CASE fb_state_entry.i16_step OF
	INIT_OBJ:	(* Zylindertyp feststellen *)
		IF st_config.b_config_fertig THEN
			(* Anzahl Spulen *)
			i16_anzahl_spulen := STRING_TO_INT(MID(st_config.str_zylinder_typ, 1, 1));
			(* Anzahl Sensoren *)
			i16_anzahl_sensoren := STRING_TO_INT(MID(st_config.str_zylinder_typ, 1, 3));
			(* Zylinder ist nockengesteuert *)
			IF FIND(st_config.str_zylinder_typ, 'NO') = 0 THEN
				b_nockengesteuert := FALSE;
			ELSE
				b_nockengesteuert := TRUE;
			END_IF
			(* Zylinder ist mit Totzeitkompensation *)
			IF FIND(st_config.str_zylinder_typ, 'TZK') = 0 THEN
				b_mit_tzk := FALSE;
			ELSE
				b_mit_tzk := TRUE;
			END_IF
			(* Vorhandene Sensoren *)
			IF FIND(st_config.str_zylinder_typ, 'AUS') >= 5 THEN
				b_sensor_ausgefahren_vorhanden := TRUE;
			ELSE
				b_sensor_ausgefahren_vorhanden := FALSE;
			END_IF
			IF FIND(st_config.str_zylinder_typ, 'EIN') >= 5 THEN
				b_sensor_eingefahren_vorhanden := TRUE;
			ELSE
				b_sensor_eingefahren_vorhanden := FALSE;
			END_IF
			fb_state_entry.i16_next_step := ZYL_INIT;
		END_IF

(*=======================================================*)
	ZYL_INIT:
		IF fb_state_entry.E THEN
			fb_ton_uz_fahren.IN := FALSE;
			fb_ton_uz_endlage1.IN := FALSE;
			fb_ton_uz_endlage2.IN := FALSE;
			fb_ton_uz_endlage3.IN := FALSE;
			fb_ton_uz_sensor1.IN := FALSE;
			fb_ton_uz_sensor2.IN := FALSE;
			fb_ton_uz_sensor3.IN := FALSE;
			st_tzk.fb_ton_tzk.IN	 := FALSE;
			fb_ton_einausfahren.IN := FALSE;
			fb_ton_quitt.IN := FALSE;
			a_ventil_ausfahren := FALSE;
			a_ventil_einfahren	:= FALSE;
			st_ctrl_out.b_fehler := FALSE;
			st_ctrl_out.b_eingefahren := FALSE;
			st_ctrl_out.b_ausgefahren := FALSE;
			st_ctrl_out.b_gestoppt := FALSE;
			st_ctrl_out.b_ohne_luft := FALSE;
			st_sm.b_zeit_ausfahren1:= FALSE;
			st_sm.b_zeit_einfahren1:= FALSE;
			st_sm.b_endlage1	:= FALSE;
			st_sm.b_sensor1:= FALSE;
			st_sm.b_zeit_ausfahren2 := FALSE;
			st_sm.b_zeit_einfahren2 := FALSE;
			st_sm.b_endlage2	:= FALSE;
			st_sm.b_sensor2 := FALSE;
			st_sm.b_zeit_ausfahren3 := FALSE;
			st_sm.b_zeit_einfahren3 := FALSE;
			st_sm.b_endlage3	:= FALSE;
			st_sm.b_sensor3 := FALSE;
			st_sm.b_winkel_ausfahren1:= FALSE;
			st_sm.b_winkel_einfahren1:= FALSE;
			st_sm.b_winkel_ausfahren2 := FALSE;
			st_sm.b_winkel_einfahren2 := FALSE;
			st_sm.b_winkel_ausfahren3 := FALSE;
			st_sm.b_winkel_einfahren3 := FALSE;
			st_sm.b_zyltyp_nicht_definiert := FALSE;
			st_sm.b_reserve1:= FALSE;
			b_direkttaste_ausfahren := FALSE;
			b_direkttaste_mittefahren := FALSE;
			b_direkttaste_einfahren	 := FALSE;
			b_zustand_uw_nocken_einfahren := FALSE;
			b_zustand_uw_nocken_ausfahren := FALSE;
		END_IF

		(*-----------------------Weiterschaltbedingungen----------------------------*)
		IF e_druckwaechter THEN
			CASE i16_anzahl_sensoren OF
			0:
				fb_state_entry.i16_next_step := GESTOPPT;

			1:
				IF b_nockengesteuert THEN
					IF bw_nocken_zylinder_einfahren THEN
						fb_state_entry.i16_next_step := BEWEGUNG_EINFAHREN;
					ELSIF bw_nocken_zylinder_ausfahren THEN
						fb_state_entry.i16_next_step := BEWEGUNG_AUSFAHREN;
					ELSE
						fb_state_entry.i16_next_step := GESTOPPT;
					END_IF
				ELSE
					IF  b_sensor_ausgefahren_vorhanden THEN
						IF NOT e_sensor1_ausgefahren THEN
							fb_state_entry.i16_next_step := BEWEGUNG_EINFAHREN;
						ELSIF e_sensor1_ausgefahren THEN
							fb_state_entry.i16_next_step := BEWEGUNG_AUSFAHREN;
						ELSE
							fb_state_entry.i16_next_step := GESTOPPT;
						END_IF
					ELSIF  b_sensor_eingefahren_vorhanden THEN
						IF e_sensor1_eingefahren THEN
							fb_state_entry.i16_next_step := BEWEGUNG_EINFAHREN;
						ELSIF NOT e_sensor1_eingefahren THEN
							fb_state_entry.i16_next_step := BEWEGUNG_AUSFAHREN;
						ELSE
							fb_state_entry.i16_next_step := GESTOPPT;
						END_IF
					END_IF
				END_IF

			2:
				IF b_nockengesteuert THEN
					IF bw_nocken_zylinder_einfahren THEN
						fb_state_entry.i16_next_step := BEWEGUNG_EINFAHREN;
					ELSIF bw_nocken_zylinder_ausfahren THEN
						fb_state_entry.i16_next_step := BEWEGUNG_AUSFAHREN;
					ELSE
						fb_state_entry.i16_next_step := GESTOPPT;
					END_IF
				ELSE
					IF b_sensor_eingefahren_vorhanden AND b_sensor_ausgefahren_vorhanden THEN
						IF e_sensor1_eingefahren THEN
							fb_state_entry.i16_next_step := BEWEGUNG_EINFAHREN;
						ELSIF e_sensor1_ausgefahren THEN
							fb_state_entry.i16_next_step := BEWEGUNG_AUSFAHREN;
						ELSE
							fb_state_entry.i16_next_step := GESTOPPT;
						END_IF
					ELSIF b_sensor_ausgefahren_vorhanden THEN
						IF NOT e_sensor1_ausgefahren AND NOT  e_sensor2_ausgefahren THEN
							fb_state_entry.i16_next_step := BEWEGUNG_EINFAHREN;
						ELSIF e_sensor1_ausgefahren OR e_sensor2_ausgefahren THEN
							fb_state_entry.i16_next_step := BEWEGUNG_AUSFAHREN;
						ELSE
							fb_state_entry.i16_next_step := GESTOPPT;
						END_IF
					ELSIF b_sensor_eingefahren_vorhanden THEN
						IF e_sensor1_eingefahren OR  e_sensor2_eingefahren THEN
							fb_state_entry.i16_next_step := BEWEGUNG_EINFAHREN;
						ELSIF NOT e_sensor1_eingefahren AND NOT e_sensor2_eingefahren THEN
							fb_state_entry.i16_next_step := BEWEGUNG_AUSFAHREN;
						ELSE
							fb_state_entry.i16_next_step := GESTOPPT;
						END_IF
					END_IF
				END_IF

			3:
				IF b_nockengesteuert THEN
					IF bw_nocken_zylinder_einfahren THEN
						fb_state_entry.i16_next_step := BEWEGUNG_EINFAHREN;
					ELSIF bw_nocken_zylinder_ausfahren THEN
						fb_state_entry.i16_next_step := BEWEGUNG_AUSFAHREN;
					ELSE
						fb_state_entry.i16_next_step := GESTOPPT;
					END_IF
				ELSE
					IF e_sensor1_eingefahren THEN
						fb_state_entry.i16_next_step := BEWEGUNG_EINFAHREN;
					ELSIF e_sensor1_ausgefahren THEN
						fb_state_entry.i16_next_step := BEWEGUNG_AUSFAHREN;
					ELSE
						fb_state_entry.i16_next_step := GESTOPPT;
					END_IF
				END_IF

			4:
				IF b_nockengesteuert THEN
					IF bw_nocken_zylinder_einfahren THEN
						fb_state_entry.i16_next_step := BEWEGUNG_EINFAHREN;
					ELSIF bw_nocken_zylinder_ausfahren THEN
						fb_state_entry.i16_next_step := BEWEGUNG_AUSFAHREN;
					ELSE
						fb_state_entry.i16_next_step := GESTOPPT;
					END_IF
				ELSE
					IF e_sensor1_eingefahren AND e_sensor2_eingefahren THEN
						fb_state_entry.i16_next_step := BEWEGUNG_EINFAHREN;
					ELSIF e_sensor1_ausgefahren AND e_sensor2_ausgefahren THEN
						fb_state_entry.i16_next_step := BEWEGUNG_AUSFAHREN;
					ELSE
						fb_state_entry.i16_next_step := GESTOPPT;
					END_IF
				END_IF

			6:
				IF b_nockengesteuert THEN
					IF bw_nocken_zylinder_einfahren THEN
						fb_state_entry.i16_next_step := BEWEGUNG_EINFAHREN;
					ELSIF bw_nocken_zylinder_ausfahren THEN
						fb_state_entry.i16_next_step := BEWEGUNG_AUSFAHREN;
					ELSE
						fb_state_entry.i16_next_step := GESTOPPT;
					END_IF
				ELSE
					IF e_sensor1_eingefahren AND e_sensor2_eingefahren AND e_sensor3_eingefahren THEN
						fb_state_entry.i16_next_step := BEWEGUNG_EINFAHREN;
					ELSIF e_sensor1_ausgefahren AND e_sensor2_ausgefahren AND e_sensor3_ausgefahren THEN
						fb_state_entry.i16_next_step := BEWEGUNG_AUSFAHREN;
					ELSE
						fb_state_entry.i16_next_step := GESTOPPT;
					END_IF
				END_IF
			END_CASE
		END_IF

(*=======================================================*)
	GESTOPPT:
		IF fb_state_entry.E THEN
			a_ventil_ausfahren := FALSE;
			a_ventil_einfahren	:= FALSE;
			st_ctrl_out.b_gestoppt := TRUE;
			st_ctrl_out.b_eingefahren := FALSE;
			st_ctrl_out.b_ausgefahren := FALSE;
			st_ctrl_out.b_ohne_luft := FALSE;
			st_ctrl_out.b_fehler := FALSE;
			b_zustand_uw_nocken_einfahren := FALSE;
			b_zustand_uw_nocken_ausfahren := FALSE;
		END_IF

		(*-----------------------Weiterschaltbedingungen----------------------------*)
		CASE i16_betriebsart OF
		KEINE:
			;
		AUTO, TIPPEN, DUMMY, PSEUDO:
			IF 	(st_ctrl_in.b_ausfahren AND
				NOT bw_nocken_zylinder_ausfahren AND
				NOT b_ibn_zylinder_ausfahren AND
				NOT b_direkttaste_ausfahren AND
				NOT e_taste_ausfahren) OR
				(NOT st_ctrl_in.b_ausfahren AND
				bw_nocken_zylinder_ausfahren AND
				NOT b_ibn_zylinder_ausfahren AND
				NOT b_direkttaste_ausfahren AND
				NOT e_taste_ausfahren) OR
				(NOT st_ctrl_in.b_ausfahren AND
				NOT bw_nocken_zylinder_ausfahren AND
				b_ibn_zylinder_ausfahren AND
				NOT b_direkttaste_ausfahren AND
				NOT e_taste_ausfahren)
				THEN
					fb_state_entry.i16_next_step := BEWEGUNG_AUSFAHREN;

			ELSIF	(st_ctrl_in.b_einfahren AND
					NOT bw_nocken_zylinder_einfahren AND
					NOT b_ibn_zylinder_einfahren AND
					NOT b_direkttaste_einfahren AND
					NOT e_taste_einfahren) OR
					(NOT st_ctrl_in.b_einfahren AND
					bw_nocken_zylinder_einfahren AND
					NOT b_ibn_zylinder_einfahren AND
					NOT b_direkttaste_einfahren AND
					NOT e_taste_einfahren) OR
					(NOT st_ctrl_in.b_einfahren AND
					NOT bw_nocken_zylinder_einfahren AND
					b_ibn_zylinder_einfahren AND
					NOT b_direkttaste_einfahren AND
					NOT e_taste_einfahren)
					THEN
						fb_state_entry.i16_next_step := BEWEGUNG_EINFAHREN;

			ELSIF	st_ctrl_in.b_luftlos AND
					NOT bw_nocken_zylinder_einfahren AND
					NOT b_ibn_zylinder_einfahren AND
					NOT b_direkttaste_einfahren AND
					NOT e_taste_einfahren AND
					NOT bw_nocken_zylinder_ausfahren AND
					NOT b_ibn_zylinder_ausfahren AND
					NOT b_direkttaste_ausfahren AND
					NOT e_taste_ausfahren
					THEN
						fb_state_entry.i16_next_step := LUFTLOS;
			END_IF
		HAND:
			IF	(st_visu.i16_nr_zyl_im_handbetrieb = st_config.i16_identnummer AND (st_visu.b_taste_ausfahren OR e_taste_ausfahren)) OR
				(bw_nocken_zylinder_ausfahren AND b_nockengesteuert AND b_masterachse_hand_dialog_aktiv)
				THEN
					fb_state_entry.i16_next_step := BEWEGUNG_AUSFAHREN;

			ELSIF	(st_visu.i16_nr_zyl_im_handbetrieb = st_config.i16_identnummer AND (st_visu.b_taste_einfahren OR e_taste_einfahren)) OR
					(bw_nocken_zylinder_einfahren AND b_nockengesteuert AND b_masterachse_hand_dialog_aktiv)
					THEN
						fb_state_entry.i16_next_step := BEWEGUNG_EINFAHREN;
			END_IF
		END_CASE

(*=======================================================*)
	EINGEFAHREN:
		IF fb_state_entry.E THEN
			st_ctrl_out.b_gestoppt := FALSE;
			st_ctrl_out.b_ausgefahren := FALSE;
			st_ctrl_out.b_ohne_luft := FALSE;
			fb_ton_einausfahren.IN := FALSE;
			fb_ton_uz_fahren.IN := FALSE;
			fb_ton_uz_sensor1.IN := FALSE;
			fb_ton_uz_sensor2.IN := FALSE;
			fb_ton_uz_sensor3.IN := FALSE;
			st_tzk.fb_ton_tzk.IN := FALSE;
			a_ventil_einfahren := TRUE;
			b_zustand_uw_nocken_einfahren := FALSE;
			IF NOT b_mit_tzk THEN
				st_ctrl_out.b_eingefahren := TRUE;
			END_IF
		END_IF

		IF st_ctrl_in.b_einfahren THEN	(* Messagewiederholung wenn der Zylinder sich schon im gewünschten Zustand befindet*)
			st_ctrl_out.b_eingefahren := TRUE;
		END_IF
	
		(*-----------------------Weiterschaltbedingungen----------------------------*)
		CASE i16_betriebsart OF
		KEINE:
			;
		AUTO, TIPPEN, DUMMY, PSEUDO:
			IF 	(st_ctrl_in.b_ausfahren AND
				NOT bw_nocken_zylinder_ausfahren AND
				NOT b_ibn_zylinder_ausfahren AND
				NOT b_direkttaste_ausfahren AND
				NOT e_taste_ausfahren) OR
				(NOT st_ctrl_in.b_ausfahren AND
				bw_nocken_zylinder_ausfahren  AND
				NOT b_ibn_zylinder_ausfahren AND
				NOT b_direkttaste_ausfahren AND
				NOT e_taste_ausfahren) OR
				(NOT st_ctrl_in.b_ausfahren AND
				NOT bw_nocken_zylinder_ausfahren AND
				b_ibn_zylinder_ausfahren AND
				NOT b_direkttaste_ausfahren AND
				NOT e_taste_ausfahren)
				THEN
					IF i16_anzahl_sensoren >= 1AND b_sensor_ausgefahren_vorhanden AND b_mit_tzk THEN
						st_tzk.t_ausfahrzeit_kompensiert := (st_tzk.t_ausfahrzeit * st_config.i16_tzk_faktor_ausfahren) / 100;
					END_IF
					fb_state_entry.i16_next_step := BEWEGUNG_AUSFAHREN;

			ELSIF	st_ctrl_in.b_luftlos AND
					NOT bw_nocken_zylinder_einfahren AND
					NOT b_ibn_zylinder_einfahren AND
					NOT b_direkttaste_einfahren AND
					NOT e_taste_einfahren AND
					NOT bw_nocken_zylinder_ausfahren AND
					NOT b_ibn_zylinder_ausfahren AND
					NOT b_direkttaste_ausfahren AND
					NOT e_taste_ausfahren
					THEN
						fb_state_entry.i16_next_step := LUFTLOS;
			END_IF
		HAND:
			IF	(st_visu.i16_nr_zyl_im_handbetrieb = st_config.i16_identnummer AND (st_visu.b_taste_ausfahren OR e_taste_ausfahren)) OR
				(bw_nocken_zylinder_ausfahren AND b_nockengesteuert AND b_masterachse_hand_dialog_aktiv)
				THEN
					IF i16_anzahl_sensoren >= 1AND b_sensor_ausgefahren_vorhanden AND b_mit_tzk THEN
						st_tzk.t_ausfahrzeit_kompensiert := (st_tzk.t_ausfahrzeit * st_config.i16_tzk_faktor_ausfahren) / 100;
					END_IF
					fb_state_entry.i16_next_step := BEWEGUNG_AUSFAHREN;
			END_IF
		END_CASE

		(* Überwachung auf Endlagenfehler *)
		IF i16_betriebsart <> HAND AND st_config.b_aktiv THEN
			CASE i16_anzahl_sensoren OF
				1,2,3:	(* Alle Zylinder mit mindestens einem Sensor für EINGEFAHREN *)
					IF b_sensor_eingefahren_vorhanden AND	st_config.b_endlage1_aktiv AND NOT e_sensor1_eingefahren THEN
						fb_ton_uz_endlage1.IN := TRUE;
						IF fb_ton_uz_endlage1.Q THEN
							st_sm.b_endlage1 := TRUE;
							fb_state_entry.i16_next_step := ZYL_FEHLER;
						END_IF
					ELSE
						fb_ton_uz_endlage1.IN := FALSE;
					END_IF
	
				4:	(* Alle Zylinder mit 2 Sensoren für EINGEFAHREN *)
					IF b_sensor_eingefahren_vorhanden AND st_config.b_endlage1_aktiv AND NOT e_sensor1_eingefahren THEN
						fb_ton_uz_endlage1.IN := TRUE;
						IF fb_ton_uz_endlage1.Q THEN
							st_sm.b_endlage1 := TRUE;
							fb_state_entry.i16_next_step := ZYL_FEHLER;
						END_IF
					ELSE
						fb_ton_uz_endlage1.IN := FALSE;
					END_IF
					IF b_sensor_eingefahren_vorhanden AND st_config.b_endlage2_aktiv AND NOT e_sensor2_eingefahren THEN
						fb_ton_uz_endlage2.IN := TRUE;
						IF fb_ton_uz_endlage2.Q THEN
							st_sm.b_endlage2 := TRUE;
							fb_state_entry.i16_next_step := ZYL_FEHLER;
						END_IF
					ELSE
						fb_ton_uz_endlage2.IN := FALSE;
					END_IF
	
				6:	(* Alle Zylinder mit 3 Sensoren für EINGEFAHREN *)
					IF b_sensor_eingefahren_vorhanden AND st_config.b_endlage1_aktiv AND NOT e_sensor1_eingefahren THEN
						fb_ton_uz_endlage1.IN := TRUE;
						IF fb_ton_uz_endlage1.Q THEN
							st_sm.b_endlage1 := TRUE;
							fb_state_entry.i16_next_step := ZYL_FEHLER;
						END_IF
					ELSE
						fb_ton_uz_endlage1.IN := FALSE;
					END_IF
					IF b_sensor_eingefahren_vorhanden AND st_config.b_endlage2_aktiv AND NOT e_sensor2_eingefahren THEN
						fb_ton_uz_endlage2.IN := TRUE;
						IF fb_ton_uz_endlage2.Q THEN
							st_sm.b_endlage2 := TRUE;
							fb_state_entry.i16_next_step := ZYL_FEHLER;
						END_IF
					ELSE
						fb_ton_uz_endlage2.IN := FALSE;
					END_IF
					IF b_sensor_eingefahren_vorhanden AND st_config.b_endlage3_aktiv AND NOT e_sensor3_eingefahren THEN
						fb_ton_uz_endlage3.IN := TRUE;
						IF fb_ton_uz_endlage3.Q THEN
							st_sm.b_endlage3 := TRUE;
							fb_state_entry.i16_next_step := ZYL_FEHLER;
						END_IF
					ELSE
						fb_ton_uz_endlage3.IN := FALSE;
					END_IF
			END_CASE
		END_IF

(*=======================================================*)
	BEWEGUNG_AUSFAHREN:
		IF fb_state_entry.E THEN
			st_ctrl_out.b_gestoppt := FALSE;
			st_ctrl_out.b_eingefahren := FALSE;
			st_ctrl_out.b_ausgefahren := FALSE;
			st_ctrl_out.b_ohne_luft := FALSE;
			st_ctrl_out.b_fehler := FALSE;
			a_ventil_einfahren := FALSE;
			a_ventil_ausfahren := TRUE;
			fb_ton_uz_fahren.IN := TRUE;
			fb_ton_einausfahren.IN := TRUE;
			fb_ton_uz_endlage1.IN := FALSE;
			fb_ton_uz_endlage2.IN := FALSE;
			fb_ton_uz_endlage3.IN := FALSE;
			st_sm.b_zeit_ausfahren1:= FALSE;
			st_sm.b_zeit_einfahren1:= FALSE;
			st_sm.b_endlage1	:= FALSE;
			st_sm.b_sensor1:= FALSE;
			st_sm.b_zeit_ausfahren2 := FALSE;
			st_sm.b_zeit_einfahren2 := FALSE;
			st_sm.b_endlage2	:= FALSE;
			st_sm.b_sensor2 := FALSE;
			st_sm.b_zeit_ausfahren3 := FALSE;
			st_sm.b_zeit_einfahren3 := FALSE;
			st_sm.b_endlage3	:= FALSE;
			st_sm.b_sensor3 := FALSE;
			st_sm.b_winkel_ausfahren1:= FALSE;
			st_sm.b_winkel_einfahren1:= FALSE;
			st_sm.b_winkel_ausfahren2 := FALSE;
			st_sm.b_winkel_einfahren2 := FALSE;
			st_sm.b_winkel_ausfahren3 := FALSE;
			st_sm.b_winkel_einfahren3 := FALSE;
			st_sm.b_zyltyp_nicht_definiert := FALSE;
			st_sm.b_reserve1:= FALSE;
			(* Verhindere die sofortige Fehlerauslösung, wenn Überwachungsnocken bei Stateentry schon vorhanden ist *)
			IF uw_nocken_zylinder_ausfahren THEN
				b_zustand_uw_nocken_ausfahren := TRUE;
			END_IF
		END_IF

		(* Fehlermeldung für nockengesteuerte Zylinder wieder freischalten *)
		IF fb_ton_uz_fahren.Q THEN
			b_zustand_uw_nocken_ausfahren := FALSE;
		END_IF

		CASE i16_betriebsart OF
		KEINE:
			;
		AUTO, TIPPEN, DUMMY, PSEUDO:
			IF	(st_ctrl_in.b_einfahren AND
				NOT bw_nocken_zylinder_einfahren AND
				NOT b_ibn_zylinder_einfahren AND
				NOT b_direkttaste_einfahren AND
				NOT e_taste_einfahren) OR
				(NOT st_ctrl_in.b_einfahren AND
				bw_nocken_zylinder_einfahren AND
				NOT b_ibn_zylinder_einfahren AND
				NOT b_direkttaste_einfahren AND
				NOT e_taste_einfahren) OR
				(NOT st_ctrl_in.b_einfahren AND
				NOT bw_nocken_zylinder_einfahren AND
				b_ibn_zylinder_einfahren AND
				NOT b_direkttaste_einfahren AND
				NOT e_taste_einfahren)
				THEN
					IF i16_anzahl_sensoren >= 1AND b_sensor_eingefahren_vorhanden AND b_mit_tzk THEN
						st_tzk.t_einfahrzeit_kompensiert := (st_tzk.t_einfahrzeit * st_config.i16_tzk_faktor_einfahren) / 100;
					END_IF
					fb_state_entry.i16_next_step := BEWEGUNG_EINFAHREN;
			END_IF
		HAND:
			IF	(st_visu.i16_nr_zyl_im_handbetrieb = st_config.i16_identnummer AND (st_visu.b_taste_einfahren OR e_taste_einfahren)) OR
				(bw_nocken_zylinder_einfahren AND b_nockengesteuert AND b_masterachse_hand_dialog_aktiv)
				THEN
					IF i16_anzahl_sensoren >= 1AND b_sensor_eingefahren_vorhanden AND b_mit_tzk THEN
						st_tzk.t_einfahrzeit_kompensiert := (st_tzk.t_einfahrzeit * st_config.i16_tzk_faktor_einfahren) / 100;
					END_IF
					fb_state_entry.i16_next_step := BEWEGUNG_EINFAHREN;
			END_IF
		END_CASE

		(* Totzeitkompensation mit Plausibilitätscheck der ermittelten Kompensationszeit *)
		IF	i16_anzahl_sensoren >= 1AND
			b_mit_tzk AND
			b_sensor_ausgefahren_vorhanden AND
			st_tzk.t_ausfahrzeit_kompensiert < st_tzk.t_ausfahrzeit
			THEN
				st_tzk.fb_ton_tzk.PT := st_tzk.t_ausfahrzeit_kompensiert ;
				st_tzk.fb_ton_tzk.IN := TRUE;
				(* Totzeit ist abgelaufen -> vorzeitig "ausgefahren" melden*)
				IF st_tzk.fb_ton_tzk.Q THEN
					st_ctrl_out.b_ausgefahren := TRUE;
				END_IF
		END_IF

		(*-----------------------Weiterschaltbedingungen----------------------------*)
		(* Bedingungen für Zylinder ist ausgefahren und Fehlervorkommen*)
		(* Die Sensorkonfiguration "vorhanden" ist nur für die Fälle 1, 2 von Bedeutung wegen Sonderzylinder *)
		CASE i16_anzahl_sensoren OF
			0:
				IF fb_ton_einausfahren.Q THEN
					fb_state_entry.i16_next_step := AUSGEFAHREN;
				END_IF

			1:
				IF b_sensor_ausgefahren_vorhanden THEN
					IF e_sensor1_ausgefahren THEN
						fb_state_entry.i16_next_step := AUSGEFAHREN;
					ELSE
						IF i16_betriebsart <> HAND AND st_config.b_aktiv THEN
							(* Zeitüberwachung *)
							IF fb_ton_uz_fahren.Q AND (NOT b_nockengesteuert OR b_no_gesteuert_im_norm_betrieb) THEN
								st_sm.b_zeit_ausfahren1 := TRUE;
								fb_state_entry.i16_next_step := ZYL_FEHLER;
							(* Winkelüberwachung *)
							ELSIF uw_nocken_zylinder_ausfahren AND b_nockengesteuert AND NOT b_no_gesteuert_im_norm_betrieb AND NOT b_zustand_uw_nocken_ausfahren THEN
								st_sm.b_winkel_ausfahren1 := TRUE;
								fb_state_entry.i16_next_step := ZYL_FEHLER;
							END_IF
						END_IF
					END_IF
				ELSIF b_sensor_eingefahren_vorhanden THEN
					IF  NOT e_sensor1_eingefahren THEN
						fb_state_entry.i16_next_step := AUSGEFAHREN;
					ELSE
						IF i16_betriebsart <> HAND AND st_config.b_aktiv THEN
							(* Zeitüberwachung *)
							IF fb_ton_uz_fahren.Q AND (NOT b_nockengesteuert OR b_no_gesteuert_im_norm_betrieb) THEN
								st_sm.b_zeit_ausfahren1 := TRUE;
								fb_state_entry.i16_next_step := ZYL_FEHLER;
							(* Winkelüberwachung *)
							ELSIF uw_nocken_zylinder_ausfahren AND b_nockengesteuert AND NOT b_no_gesteuert_im_norm_betrieb AND NOT b_zustand_uw_nocken_ausfahren THEN
								st_sm.b_winkel_ausfahren1 := TRUE;
								fb_state_entry.i16_next_step := ZYL_FEHLER;
							END_IF
						END_IF
					END_IF
				END_IF

			2:
				IF b_sensor_eingefahren_vorhanden AND b_sensor_ausgefahren_vorhanden THEN
					IF e_sensor1_ausgefahren AND NOT e_sensor1_eingefahren THEN
						fb_state_entry.i16_next_step := AUSGEFAHREN;
					ELSE
						IF i16_betriebsart <> HAND AND st_config.b_aktiv THEN
							(* Zeitüberwachung *)
							IF fb_ton_uz_fahren.Q AND (NOT b_nockengesteuert OR b_no_gesteuert_im_norm_betrieb) THEN
								st_sm.b_zeit_ausfahren1 := TRUE;
								fb_state_entry.i16_next_step := ZYL_FEHLER;
							(* Winkelüberwachung *)
							ELSIF uw_nocken_zylinder_ausfahren AND b_nockengesteuert AND NOT b_no_gesteuert_im_norm_betrieb AND NOT b_zustand_uw_nocken_ausfahren THEN
								st_sm.b_winkel_ausfahren1 := TRUE;
								fb_state_entry.i16_next_step := ZYL_FEHLER;
							END_IF
						END_IF
					END_IF
				ELSIF b_sensor_eingefahren_vorhanden THEN
					IF NOT e_sensor1_eingefahren AND NOT e_sensor2_eingefahren THEN
						fb_state_entry.i16_next_step := AUSGEFAHREN;
					ELSE
						IF i16_betriebsart <> HAND AND st_config.b_aktiv THEN
							(* Zeitüberwachung *)
							IF fb_ton_uz_fahren.Q AND (NOT b_nockengesteuert OR b_no_gesteuert_im_norm_betrieb) THEN
								IF e_sensor1_eingefahren THEN
									st_sm.b_zeit_ausfahren1 := TRUE;
								END_IF
								IF e_sensor2_eingefahren THEN
									st_sm.b_zeit_ausfahren2 := TRUE;
								END_IF
								fb_state_entry.i16_next_step := ZYL_FEHLER;
							(* Winkelüberwachung *)
							ELSIF uw_nocken_zylinder_ausfahren AND b_nockengesteuert AND NOT b_no_gesteuert_im_norm_betrieb AND NOT b_zustand_uw_nocken_ausfahren THEN
								IF e_sensor1_eingefahren THEN
									st_sm.b_winkel_ausfahren1 := TRUE;
								END_IF
								IF e_sensor2_eingefahren THEN
									st_sm.b_winkel_ausfahren2 := TRUE;
								END_IF
								fb_state_entry.i16_next_step := ZYL_FEHLER;
							END_IF
						END_IF
					END_IF
				ELSIF  b_sensor_ausgefahren_vorhanden THEN
					IF e_sensor1_ausgefahren AND e_sensor2_ausgefahren THEN
						fb_state_entry.i16_next_step := AUSGEFAHREN;
					ELSE
						IF i16_betriebsart <> HAND AND st_config.b_aktiv THEN
							(* Zeitüberwachung *)
							IF fb_ton_uz_fahren.Q AND (NOT b_nockengesteuert OR b_no_gesteuert_im_norm_betrieb) THEN
								IF NOT e_sensor1_ausgefahren THEN
									st_sm.b_zeit_ausfahren1 := TRUE;
								END_IF
								IF NOT e_sensor2_ausgefahren THEN
									st_sm.b_zeit_ausfahren2 := TRUE;
								END_IF
								fb_state_entry.i16_next_step := ZYL_FEHLER;
							(* Winkelüberwachung *)
							ELSIF uw_nocken_zylinder_ausfahren AND b_nockengesteuert AND NOT b_no_gesteuert_im_norm_betrieb AND NOT b_zustand_uw_nocken_ausfahren THEN
								IF NOT e_sensor1_ausgefahren THEN
									st_sm.b_winkel_ausfahren1 := TRUE;
								END_IF
								IF NOT e_sensor2_ausgefahren THEN
									st_sm.b_winkel_ausfahren2 := TRUE;
								END_IF
								fb_state_entry.i16_next_step := ZYL_FEHLER;
							END_IF
						END_IF
					END_IF
				END_IF
				IF i16_betriebsart <> HAND AND st_config.b_aktiv THEN
					(* Überwachung auf Sensorfehler *)
					IF e_sensor1_ausgefahren  AND e_sensor1_eingefahren  AND st_config.b_sensor1_aktiv THEN
						fb_ton_uz_sensor1.IN := TRUE;
						IF fb_ton_uz_sensor1.Q THEN
							st_sm.b_sensor1 := TRUE;
							fb_state_entry.i16_next_step := ZYL_FEHLER;
						END_IF
					ELSE
						fb_ton_uz_sensor1.IN := FALSE;
					END_IF
				END_IF

			3:
				IF	(* Zylinder ist ausgefahren *)
					(e_sensor1_ausgefahren AND NOT e_sensor1_eingefahren AND NOT e_sensor_mittegefahren) OR
					(* Zylinder steht in Mittelstellung *)
					(e_sensor_mittegefahren AND NOT e_sensor1_eingefahren AND NOT e_sensor1_ausgefahren)
					THEN
						fb_state_entry.i16_next_step := AUSGEFAHREN;
				ELSE
					IF i16_betriebsart <> HAND AND st_config.b_aktiv THEN
						(* Zeitüberwachung *)
						IF fb_ton_uz_fahren.Q AND (NOT b_nockengesteuert OR b_no_gesteuert_im_norm_betrieb) THEN
							st_sm.b_zeit_ausfahren1 := TRUE;
							fb_state_entry.i16_next_step := ZYL_FEHLER;
						(* Winkelüberwachung *)
						ELSIF uw_nocken_zylinder_ausfahren AND b_nockengesteuert AND NOT b_no_gesteuert_im_norm_betrieb AND NOT b_zustand_uw_nocken_ausfahren THEN
							st_sm.b_winkel_ausfahren1 := TRUE;
							fb_state_entry.i16_next_step := ZYL_FEHLER;
						END_IF
					END_IF
				END_IF
				IF i16_betriebsart <> HAND AND st_config.b_aktiv THEN
					(* Überwachung auf Sensorfehler *)
					IF e_sensor1_ausgefahren  AND e_sensor1_eingefahren  AND st_config.b_sensor1_aktiv THEN
						fb_ton_uz_sensor1.IN := TRUE;
						IF fb_ton_uz_sensor1.Q THEN
							st_sm.b_sensor1 := TRUE;
							fb_state_entry.i16_next_step := ZYL_FEHLER;
						END_IF
					ELSE
						fb_ton_uz_sensor1.IN := FALSE;
					END_IF
				END_IF

			4:
				IF e_sensor1_ausgefahren AND e_sensor2_ausgefahren AND NOT e_sensor1_eingefahren AND NOT e_sensor2_eingefahren	THEN
					fb_state_entry.i16_next_step := AUSGEFAHREN;
				ELSE
					IF i16_betriebsart <> HAND AND st_config.b_aktiv THEN
						IF NOT e_sensor1_ausgefahren OR NOT e_sensor2_ausgefahren THEN
							(* Zeitüberwachung *)
							IF fb_ton_uz_fahren.Q AND (NOT b_nockengesteuert OR b_no_gesteuert_im_norm_betrieb) THEN
								IF NOT e_sensor1_ausgefahren THEN
									st_sm.b_zeit_ausfahren1 := TRUE;
								END_IF
								IF NOT e_sensor2_ausgefahren THEN
									st_sm.b_zeit_ausfahren2 := TRUE;
								END_IF
								fb_state_entry.i16_next_step := ZYL_FEHLER;
							(* Winkelüberwachung *)
							ELSIF uw_nocken_zylinder_ausfahren AND b_nockengesteuert AND NOT b_no_gesteuert_im_norm_betrieb AND NOT b_zustand_uw_nocken_ausfahren THEN
								IF NOT e_sensor1_ausgefahren THEN
									st_sm.b_winkel_ausfahren1 := TRUE;
								END_IF
								IF NOT e_sensor2_ausgefahren THEN
									st_sm.b_winkel_ausfahren2 := TRUE;
								END_IF
								fb_state_entry.i16_next_step := ZYL_FEHLER;
							END_IF
						END_IF
					END_IF
				END_IF

				IF i16_betriebsart <> HAND AND st_config.b_aktiv THEN
					(* Überwachung auf Sensorfehler *)
					IF e_sensor1_ausgefahren  AND e_sensor1_eingefahren  AND st_config.b_sensor1_aktiv THEN
						fb_ton_uz_sensor1.IN := TRUE;
						IF fb_ton_uz_sensor1.Q THEN
							st_sm.b_sensor1 := TRUE;
							fb_state_entry.i16_next_step := ZYL_FEHLER;
						END_IF
					ELSE
						fb_ton_uz_sensor1.IN := FALSE;
					END_IF
					IF e_sensor2_ausgefahren  AND e_sensor2_eingefahren  AND st_config.b_sensor2_aktiv THEN
						fb_ton_uz_sensor2.IN := TRUE;
						IF fb_ton_uz_sensor2.Q THEN
							st_sm.b_sensor2 := TRUE;
							fb_state_entry.i16_next_step := ZYL_FEHLER;
						END_IF
					ELSE
						fb_ton_uz_sensor2.IN := FALSE;
					END_IF
				END_IF

			6:
				IF 	e_sensor1_ausgefahren AND
					e_sensor2_ausgefahren AND
					e_sensor3_ausgefahren AND
					NOT e_sensor1_eingefahren AND
					NOT e_sensor2_eingefahren AND
					NOT e_sensor3_eingefahren
					THEN
						fb_state_entry.i16_next_step := AUSGEFAHREN;
				ELSE
					IF i16_betriebsart <> HAND AND st_config.b_aktiv THEN
						IF NOT e_sensor1_ausgefahren OR NOT e_sensor2_ausgefahren OR NOT e_sensor3_ausgefahren THEN
							(* Zeitüberwachung *)
							IF fb_ton_uz_fahren.Q AND (NOT b_nockengesteuert OR b_no_gesteuert_im_norm_betrieb) THEN
								IF NOT e_sensor1_ausgefahren THEN
									st_sm.b_zeit_ausfahren1 := TRUE;
								END_IF
								IF NOT e_sensor2_ausgefahren THEN
									st_sm.b_zeit_ausfahren2 := TRUE;
								END_IF
								IF NOT e_sensor3_ausgefahren THEN
									st_sm.b_zeit_ausfahren3 := TRUE;
								END_IF
								fb_state_entry.i16_next_step := ZYL_FEHLER;
							(* Winkelüberwachung *)
							ELSIF uw_nocken_zylinder_ausfahren AND b_nockengesteuert AND NOT b_no_gesteuert_im_norm_betrieb AND NOT b_zustand_uw_nocken_ausfahren THEN
								IF NOT e_sensor1_ausgefahren THEN
									st_sm.b_winkel_ausfahren1 := TRUE;
								END_IF
								IF NOT e_sensor2_ausgefahren THEN
									st_sm.b_winkel_ausfahren2 := TRUE;
								END_IF
								IF NOT e_sensor3_ausgefahren THEN
									st_sm.b_winkel_ausfahren3 := TRUE;
								END_IF
								fb_state_entry.i16_next_step := ZYL_FEHLER;
							END_IF
						END_IF
					END_IF
				END_IF

				IF i16_betriebsart <> HAND AND st_config.b_aktiv THEN
					(* Überwachung auf Sensorfehler *)
					IF e_sensor1_ausgefahren  AND e_sensor1_eingefahren  AND st_config.b_sensor1_aktiv THEN
						fb_ton_uz_sensor1.IN := TRUE;
						IF fb_ton_uz_sensor1.Q THEN
							st_sm.b_sensor1 := TRUE;
							fb_state_entry.i16_next_step := ZYL_FEHLER;
						END_IF
					ELSE
						fb_ton_uz_sensor1.IN := FALSE;
					END_IF
					IF e_sensor2_ausgefahren  AND e_sensor2_eingefahren  AND st_config.b_sensor2_aktiv THEN
						fb_ton_uz_sensor2.IN := TRUE;
						IF fb_ton_uz_sensor2.Q THEN
							st_sm.b_sensor2 := TRUE;
							fb_state_entry.i16_next_step := ZYL_FEHLER;
						END_IF
					ELSE
						fb_ton_uz_sensor2.IN := FALSE;
					END_IF
					IF e_sensor3_ausgefahren  AND e_sensor3_eingefahren  AND st_config.b_sensor3_aktiv THEN
						fb_ton_uz_sensor3.IN := TRUE;
						IF fb_ton_uz_sensor3.Q THEN
							st_sm.b_sensor3 := TRUE;
							fb_state_entry.i16_next_step := ZYL_FEHLER;
						END_IF
					ELSE
						fb_ton_uz_sensor3.IN := FALSE;
					END_IF
				END_IF
		END_CASE

(*=======================================================*)
	AUSGEFAHREN:
		IF fb_state_entry.E THEN
			st_ctrl_out.b_gestoppt := FALSE;
			st_ctrl_out.b_eingefahren := FALSE;
			st_ctrl_out.b_ohne_luft := FALSE;
			fb_ton_einausfahren.IN := FALSE;
			fb_ton_uz_fahren.IN := FALSE;
			fb_ton_uz_sensor1.IN := FALSE;
			fb_ton_uz_sensor2.IN := FALSE;
			fb_ton_uz_sensor3.IN := FALSE;
			st_tzk.fb_ton_tzk.IN := FALSE;
			a_ventil_ausfahren := TRUE;
			b_zustand_uw_nocken_ausfahren := FALSE;
			IF NOT b_mit_tzk THEN
				st_ctrl_out.b_ausgefahren := TRUE;
			END_IF
		END_IF

		IF st_ctrl_in.b_ausfahren THEN	(* Messagewiederholung wenn der Zylinder sich schon im gewünschten Zustand befindet*)
			st_ctrl_out.b_ausgefahren := TRUE;
		END_IF

		(*-----------------------Weiterschaltbedingungen----------------------------*)
		CASE i16_betriebsart OF
		KEINE:
			;
		AUTO, TIPPEN, DUMMY, PSEUDO:
			IF	(st_ctrl_in.b_einfahren AND
				NOT bw_nocken_zylinder_einfahren AND
				NOT b_ibn_zylinder_einfahren AND
				NOT b_direkttaste_einfahren AND
				NOT e_taste_einfahren) OR
				(NOT st_ctrl_in.b_einfahren AND
				bw_nocken_zylinder_einfahren AND
				NOT b_ibn_zylinder_einfahren AND
				NOT b_direkttaste_einfahren AND
				NOT e_taste_einfahren) OR
				(NOT st_ctrl_in.b_einfahren AND
				NOT bw_nocken_zylinder_einfahren AND
				b_ibn_zylinder_einfahren AND
				NOT b_direkttaste_einfahren AND
				NOT e_taste_einfahren)
				THEN
					IF i16_anzahl_sensoren >= 1AND b_sensor_eingefahren_vorhanden AND b_mit_tzk THEN
						st_tzk.t_einfahrzeit_kompensiert := (st_tzk.t_einfahrzeit * st_config.i16_tzk_faktor_einfahren) / 100;
					END_IF
					fb_state_entry.i16_next_step := BEWEGUNG_EINFAHREN;

			ELSIF	st_ctrl_in.b_luftlos AND
					NOT bw_nocken_zylinder_einfahren AND
					NOT b_ibn_zylinder_einfahren AND
					NOT b_direkttaste_einfahren AND
					NOT e_taste_einfahren AND
					NOT bw_nocken_zylinder_ausfahren AND
					NOT b_ibn_zylinder_ausfahren AND
					NOT b_direkttaste_ausfahren AND
					NOT e_taste_ausfahren
					THEN
						fb_state_entry.i16_next_step := LUFTLOS;
			END_IF
		HAND:
			IF	(st_visu.i16_nr_zyl_im_handbetrieb = st_config.i16_identnummer AND (st_visu.b_taste_einfahren OR e_taste_einfahren)) OR
				(bw_nocken_zylinder_einfahren AND b_nockengesteuert AND b_masterachse_hand_dialog_aktiv)
				THEN
					IF i16_anzahl_sensoren >= 1AND b_sensor_eingefahren_vorhanden AND b_mit_tzk THEN
						st_tzk.t_einfahrzeit_kompensiert := (st_tzk.t_einfahrzeit * st_config.i16_tzk_faktor_einfahren) / 100;
					END_IF
					fb_state_entry.i16_next_step := BEWEGUNG_EINFAHREN;
			END_IF
		END_CASE

		(* Überwachung auf Endlagenfehler *)
		IF i16_betriebsart <> HAND AND st_config.b_aktiv THEN
			CASE i16_anzahl_sensoren OF
				1,2,3:	(* Alle Zylinder mit mindestens einem Sensor für EINGEFAHREN *)
					IF b_sensor_ausgefahren_vorhanden AND st_config.b_endlage1_aktiv AND NOT e_sensor1_ausgefahren THEN
						fb_ton_uz_endlage1.IN := TRUE;
						IF fb_ton_uz_endlage1.Q THEN
							st_sm.b_endlage1 := TRUE;
							fb_state_entry.i16_next_step := ZYL_FEHLER;
						END_IF
					ELSE
						fb_ton_uz_endlage1.IN := FALSE;
					END_IF

				4:	(* Alle Zylinder mit 2 Sensoren für EINGEFAHREN *)
					IF b_sensor_ausgefahren_vorhanden AND st_config.b_endlage1_aktiv AND NOT e_sensor1_ausgefahren THEN
						fb_ton_uz_endlage1.IN := TRUE;
						IF fb_ton_uz_endlage1.Q THEN
							st_sm.b_endlage1 := TRUE;
							fb_state_entry.i16_next_step := ZYL_FEHLER;
						END_IF
					ELSE
						fb_ton_uz_endlage1.IN := FALSE;
					END_IF
					IF b_sensor_ausgefahren_vorhanden AND st_config.b_endlage2_aktiv AND NOT e_sensor2_ausgefahren THEN
						fb_ton_uz_endlage2.IN := TRUE;
						IF fb_ton_uz_endlage2.Q THEN
							st_sm.b_endlage2 := TRUE;
							fb_state_entry.i16_next_step := ZYL_FEHLER;
						END_IF
					ELSE
						fb_ton_uz_endlage2.IN := FALSE;
					END_IF

				6:	(* Alle Zylinder mit 3 Sensoren für EINGEFAHREN *)
					IF b_sensor_ausgefahren_vorhanden AND st_config.b_endlage1_aktiv AND NOT e_sensor1_ausgefahren THEN
						fb_ton_uz_endlage1.IN := TRUE;
						IF fb_ton_uz_endlage1.Q THEN
							st_sm.b_endlage1 := TRUE;
							fb_state_entry.i16_next_step := ZYL_FEHLER;
						END_IF
					ELSE
						fb_ton_uz_endlage1.IN := FALSE;
					END_IF
					IF b_sensor_ausgefahren_vorhanden AND st_config.b_endlage2_aktiv AND NOT e_sensor2_ausgefahren THEN
						fb_ton_uz_endlage2.IN := TRUE;
						IF fb_ton_uz_endlage2.Q THEN
							st_sm.b_endlage2 := TRUE;
							fb_state_entry.i16_next_step := ZYL_FEHLER;
						END_IF
					ELSE
						fb_ton_uz_endlage2.IN := FALSE;
					END_IF
					IF b_sensor_ausgefahren_vorhanden AND st_config.b_endlage3_aktiv AND NOT e_sensor3_ausgefahren THEN
						fb_ton_uz_endlage3.IN := TRUE;
						IF fb_ton_uz_endlage3.Q THEN
							st_sm.b_endlage3 := TRUE;
							fb_state_entry.i16_next_step := ZYL_FEHLER;
						END_IF
					ELSE
						fb_ton_uz_endlage3.IN := FALSE;
					END_IF
			END_CASE
		END_IF

(*=======================================================*)
	BEWEGUNG_EINFAHREN:
		IF fb_state_entry.E THEN
			st_ctrl_out.b_gestoppt := FALSE;
			st_ctrl_out.b_eingefahren := FALSE;
			st_ctrl_out.b_ausgefahren := FALSE;
			st_ctrl_out.b_ohne_luft := FALSE;
			st_ctrl_out.b_fehler := FALSE;
			a_ventil_ausfahren := FALSE;
			a_ventil_einfahren := TRUE;
			fb_ton_uz_fahren.IN := TRUE;
			fb_ton_einausfahren.IN := TRUE;
			fb_ton_uz_endlage1.IN := FALSE;
			fb_ton_uz_endlage2.IN := FALSE;
			fb_ton_uz_endlage3.IN := FALSE;
			st_sm.b_zeit_ausfahren1:= FALSE;
			st_sm.b_zeit_einfahren1:= FALSE;
			st_sm.b_endlage1	:= FALSE;
			st_sm.b_sensor1:= FALSE;
			st_sm.b_zeit_ausfahren2 := FALSE;
			st_sm.b_zeit_einfahren2 := FALSE;
			st_sm.b_endlage2	:= FALSE;
			st_sm.b_sensor2 := FALSE;
			st_sm.b_zeit_ausfahren3 := FALSE;
			st_sm.b_zeit_einfahren3 := FALSE;
			st_sm.b_endlage3	:= FALSE;
			st_sm.b_sensor3 := FALSE;
			st_sm.b_winkel_ausfahren1:= FALSE;
			st_sm.b_winkel_einfahren1:= FALSE;
			st_sm.b_winkel_ausfahren2 := FALSE;
			st_sm.b_winkel_einfahren2 := FALSE;
			st_sm.b_winkel_ausfahren3 := FALSE;
			st_sm.b_winkel_einfahren3 := FALSE;
			st_sm.b_zyltyp_nicht_definiert := FALSE;
			st_sm.b_reserve1:= FALSE;
			(* Verhindere die sofortige Fehlerauslösung, wenn Überwachungsnocken bei Stateentry schon vorhanden ist *)
			IF uw_nocken_zylinder_einfahren THEN
				b_zustand_uw_nocken_einfahren := TRUE;
			END_IF
		END_IF

		(* Fehlermeldung für nockengesteuerte Zylinder wieder freischalten *)
		IF fb_ton_uz_fahren.Q THEN
			b_zustand_uw_nocken_einfahren := FALSE;
		END_IF

		CASE i16_betriebsart OF
		KEINE:
			;
		AUTO, TIPPEN, DUMMY, PSEUDO:
			IF 	(st_ctrl_in.b_ausfahren AND
				NOT bw_nocken_zylinder_ausfahren AND
				NOT b_ibn_zylinder_ausfahren AND
				NOT b_direkttaste_ausfahren AND
				NOT e_taste_ausfahren) OR
				(NOT st_ctrl_in.b_ausfahren AND
				bw_nocken_zylinder_ausfahren AND
				NOT b_ibn_zylinder_ausfahren AND
				NOT b_direkttaste_ausfahren AND
				NOT e_taste_ausfahren) OR
				(NOT st_ctrl_in.b_ausfahren AND
				NOT bw_nocken_zylinder_ausfahren AND
				b_ibn_zylinder_ausfahren AND
				NOT b_direkttaste_ausfahren AND
				NOT e_taste_ausfahren)
				THEN
					IF i16_anzahl_sensoren >= 1AND b_sensor_ausgefahren_vorhanden AND b_mit_tzk THEN
						st_tzk.t_ausfahrzeit_kompensiert := (st_tzk.t_ausfahrzeit * st_config.i16_tzk_faktor_ausfahren) / 100;
					END_IF
					fb_state_entry.i16_next_step := BEWEGUNG_AUSFAHREN;
			END_IF
		HAND:
			IF	(st_visu.i16_nr_zyl_im_handbetrieb = st_config.i16_identnummer AND (st_visu.b_taste_ausfahren OR e_taste_ausfahren)) OR
				(bw_nocken_zylinder_ausfahren AND b_nockengesteuert AND b_masterachse_hand_dialog_aktiv)
				THEN
					IF i16_anzahl_sensoren >= 1AND b_sensor_ausgefahren_vorhanden AND b_mit_tzk THEN
						st_tzk.t_ausfahrzeit_kompensiert := (st_tzk.t_ausfahrzeit * st_config.i16_tzk_faktor_ausfahren) / 100;
					END_IF
					fb_state_entry.i16_next_step := BEWEGUNG_AUSFAHREN;
			END_IF
		END_CASE

		(* Totzeitkompensation mit Plausibilitätscheck der ermittelten Kompensationszeit *)
		IF 	i16_anzahl_sensoren >= 1AND
			b_sensor_eingefahren_vorhanden AND
			b_mit_tzk AND
			st_tzk.t_einfahrzeit_kompensiert < st_tzk.t_einfahrzeit
			THEN
				st_tzk.fb_ton_tzk.PT := st_tzk.t_einfahrzeit_kompensiert ;
				st_tzk.fb_ton_tzk.IN := TRUE;
				(* Totzeit ist abgelaufen -> vorzeitig "eingefahren" melden*)
				IF st_tzk.fb_ton_tzk.Q THEN
					st_tzk.fb_ton_tzk.IN := FALSE;
					st_ctrl_out.b_eingefahren := TRUE;
				END_IF
		END_IF

		(*-----------------------Weiterschaltbedingungen----------------------------*)
		(* Bedingungen für Zylinder ist eingefahren und Fehlervorkommen*)
		(* Die Sensorkonfiguration "vorhanden" ist nur für die Fälle 1, 2 von Bedeutung wegen Sonderzylinder *)
		CASE i16_anzahl_sensoren OF
			0:
				IF fb_ton_einausfahren.Q THEN
					fb_state_entry.i16_next_step := EINGEFAHREN;
				END_IF

			1:
				IF b_sensor_eingefahren_vorhanden THEN
					IF e_sensor1_eingefahren THEN
						fb_state_entry.i16_next_step := EINGEFAHREN;
					ELSE
						IF i16_betriebsart <> HAND AND st_config.b_aktiv THEN
							(* Zeitüberwachung *)
							IF fb_ton_uz_fahren.Q AND (NOT b_nockengesteuert OR b_no_gesteuert_im_norm_betrieb)THEN
								st_sm.b_zeit_einfahren1 := TRUE;
								fb_state_entry.i16_next_step := ZYL_FEHLER;
							(* Winkelüberwachung *)
							ELSIF uw_nocken_zylinder_einfahren AND b_nockengesteuert AND NOT b_no_gesteuert_im_norm_betrieb AND NOT b_zustand_uw_nocken_einfahren THEN
								st_sm.b_winkel_einfahren1 := TRUE;
								fb_state_entry.i16_next_step := ZYL_FEHLER;
							END_IF
						END_IF
					END_IF
				ELSIF b_sensor_ausgefahren_vorhanden THEN
					IF  NOT e_sensor1_ausgefahren THEN
						fb_state_entry.i16_next_step := EINGEFAHREN;
					ELSE
						IF i16_betriebsart <> HAND AND st_config.b_aktiv THEN
							(* Zeitüberwachung *)
							IF fb_ton_uz_fahren.Q AND (NOT b_nockengesteuert OR b_no_gesteuert_im_norm_betrieb)THEN
								st_sm.b_zeit_einfahren1 := TRUE;
								fb_state_entry.i16_next_step := ZYL_FEHLER;
							(* Winkelüberwachung *)
							ELSIF uw_nocken_zylinder_einfahren AND b_nockengesteuert AND NOT b_no_gesteuert_im_norm_betrieb AND NOT b_zustand_uw_nocken_einfahren THEN
								st_sm.b_winkel_einfahren1 := TRUE;
								fb_state_entry.i16_next_step := ZYL_FEHLER;
							END_IF
						END_IF
					END_IF
				END_IF

			2:
				IF b_sensor_eingefahren_vorhanden AND b_sensor_ausgefahren_vorhanden THEN
					IF e_sensor1_eingefahren AND NOT e_sensor1_ausgefahren THEN
						fb_state_entry.i16_next_step := EINGEFAHREN;
					ELSE
						IF i16_betriebsart <> HAND AND st_config.b_aktiv THEN
							(* Zeitüberwachung *)
							IF fb_ton_uz_fahren.Q AND (NOT b_nockengesteuert OR b_no_gesteuert_im_norm_betrieb)THEN
								st_sm.b_zeit_einfahren1 := TRUE;
								fb_state_entry.i16_next_step := ZYL_FEHLER;
							(* Winkelüberwachung *)
							ELSIF uw_nocken_zylinder_einfahren AND b_nockengesteuert AND NOT b_no_gesteuert_im_norm_betrieb AND NOT b_zustand_uw_nocken_einfahren THEN
								st_sm.b_winkel_einfahren1 := TRUE;
								fb_state_entry.i16_next_step := ZYL_FEHLER;
							END_IF
						END_IF
					END_IF
				ELSIF b_sensor_ausgefahren_vorhanden THEN
					IF NOT e_sensor1_ausgefahren AND NOT e_sensor2_ausgefahren THEN
						fb_state_entry.i16_next_step := EINGEFAHREN;
					ELSE
						IF i16_betriebsart <> HAND AND st_config.b_aktiv THEN
							(* Zeitüberwachung *)
							IF fb_ton_uz_fahren.Q AND (NOT b_nockengesteuert OR b_no_gesteuert_im_norm_betrieb)THEN
								IF e_sensor1_ausgefahren THEN
									st_sm.b_zeit_einfahren1 := TRUE;
								END_IF
								IF e_sensor2_ausgefahren THEN
									st_sm.b_zeit_einfahren2 := TRUE;
								END_IF
								fb_state_entry.i16_next_step := ZYL_FEHLER;
							(* Winkelüberwachung *)
							ELSIF uw_nocken_zylinder_einfahren AND b_nockengesteuert AND NOT b_no_gesteuert_im_norm_betrieb AND NOT b_zustand_uw_nocken_einfahren THEN
								IF e_sensor1_ausgefahren THEN
								st_sm.b_winkel_einfahren1 := TRUE;
								END_IF
								IF e_sensor2_ausgefahren THEN
								st_sm.b_winkel_einfahren2 := TRUE;
								END_IF
								fb_state_entry.i16_next_step := ZYL_FEHLER;
							END_IF
						END_IF
					END_IF
				ELSIF  b_sensor_eingefahren_vorhanden THEN
					IF e_sensor1_eingefahren AND e_sensor2_eingefahren THEN
						fb_state_entry.i16_next_step := EINGEFAHREN;
					ELSE
						IF i16_betriebsart <> HAND AND st_config.b_aktiv THEN
							(* Zeitüberwachung *)
							IF fb_ton_uz_fahren.Q AND (NOT b_nockengesteuert OR b_no_gesteuert_im_norm_betrieb)THEN
								IF NOT e_sensor1_eingefahren THEN
									st_sm.b_zeit_einfahren1 := TRUE;
								END_IF
								IF NOT e_sensor2_eingefahren THEN
									st_sm.b_zeit_einfahren2 := TRUE;
								END_IF
								fb_state_entry.i16_next_step := ZYL_FEHLER;
							(* Winkelüberwachung *)
							ELSIF uw_nocken_zylinder_einfahren AND b_nockengesteuert AND NOT b_no_gesteuert_im_norm_betrieb AND NOT b_zustand_uw_nocken_einfahren THEN
								IF NOT e_sensor1_eingefahren THEN
									st_sm.b_winkel_einfahren1 := TRUE;
								END_IF
								IF NOT e_sensor2_eingefahren THEN
									st_sm.b_winkel_einfahren2 := TRUE;
								END_IF
								fb_state_entry.i16_next_step := ZYL_FEHLER;
							END_IF
						END_IF
					END_IF
				END_IF
				IF i16_betriebsart <> HAND AND st_config.b_aktiv THEN
					(* Überwachung auf Sensorfehler *)
					IF e_sensor1_ausgefahren  AND e_sensor1_eingefahren  AND st_config.b_sensor1_aktiv THEN
						fb_ton_uz_sensor1.IN := TRUE;
						IF fb_ton_uz_sensor1.Q THEN
							st_sm.b_sensor1 := TRUE;
							fb_state_entry.i16_next_step := ZYL_FEHLER;
						END_IF
					ELSE
						fb_ton_uz_sensor1.IN := FALSE;
					END_IF
				END_IF

			3:
				IF	(* Zylinder ist ausgefahren *)
					(e_sensor1_eingefahren AND NOT e_sensor1_ausgefahren AND NOT e_sensor_mittegefahren) OR
					(* Zylinder steht in Mittelstellung *)
					(e_sensor_mittegefahren AND NOT e_sensor1_eingefahren AND NOT e_sensor1_ausgefahren)
					THEN
						fb_state_entry.i16_next_step := EINGEFAHREN;
				ELSE
					IF i16_betriebsart <> HAND AND st_config.b_aktiv THEN
						(* Zeitüberwachung *)
						IF fb_ton_uz_fahren.Q AND (NOT b_nockengesteuert OR b_no_gesteuert_im_norm_betrieb)THEN
							st_sm.b_zeit_einfahren1 := TRUE;
							fb_state_entry.i16_next_step := ZYL_FEHLER;
						(* Winkelüberwachung *)
						ELSIF uw_nocken_zylinder_einfahren AND b_nockengesteuert AND NOT b_no_gesteuert_im_norm_betrieb AND NOT b_zustand_uw_nocken_einfahren THEN
							st_sm.b_winkel_einfahren1 := TRUE;
							fb_state_entry.i16_next_step := ZYL_FEHLER;
						END_IF
					END_IF
				END_IF
				IF i16_betriebsart <> HAND AND st_config.b_aktiv THEN
					(* Überwachung auf Sensorfehler *)
					IF e_sensor1_ausgefahren  AND e_sensor1_eingefahren  AND st_config.b_sensor1_aktiv THEN
						fb_ton_uz_sensor1.IN := TRUE;
						IF fb_ton_uz_sensor1.Q THEN
							st_sm.b_sensor1 := TRUE;
							fb_state_entry.i16_next_step := ZYL_FEHLER;
						END_IF
					ELSE
						fb_ton_uz_sensor1.IN := FALSE;
					END_IF
				END_IF

			4:
				IF e_sensor1_eingefahren AND e_sensor2_eingefahren AND NOT e_sensor1_ausgefahren AND NOT e_sensor2_ausgefahren	THEN
					fb_state_entry.i16_next_step := EINGEFAHREN;
				ELSE
					IF i16_betriebsart <> HAND AND st_config.b_aktiv THEN
						IF NOT e_sensor1_eingefahren OR NOT e_sensor2_eingefahren THEN
							(* Zeitüberwachung *)
							IF fb_ton_uz_fahren.Q AND (NOT b_nockengesteuert OR b_no_gesteuert_im_norm_betrieb)THEN
								IF NOT e_sensor1_eingefahren THEN
									st_sm.b_zeit_einfahren1 := TRUE;
								END_IF
								IF NOT e_sensor2_eingefahren THEN
									st_sm.b_zeit_einfahren2 := TRUE;
								END_IF
								fb_state_entry.i16_next_step := ZYL_FEHLER;
							(* Winkelüberwachung *)
							ELSIF uw_nocken_zylinder_einfahren AND b_nockengesteuert AND NOT b_no_gesteuert_im_norm_betrieb AND NOT b_zustand_uw_nocken_einfahren THEN
								IF NOT e_sensor1_eingefahren THEN
									st_sm.b_winkel_einfahren1 := TRUE;
								END_IF
								IF NOT e_sensor2_eingefahren THEN
									st_sm.b_winkel_einfahren2 := TRUE;
								END_IF
								fb_state_entry.i16_next_step := ZYL_FEHLER;
							END_IF
						END_IF
					END_IF
				END_IF

				IF i16_betriebsart <> HAND AND st_config.b_aktiv THEN
					(* Überwachung auf Sensorfehler *)
					IF e_sensor1_ausgefahren  AND e_sensor1_eingefahren  AND st_config.b_sensor1_aktiv THEN
						fb_ton_uz_sensor1.IN := TRUE;
						IF fb_ton_uz_sensor1.Q THEN
							st_sm.b_sensor1 := TRUE;
							fb_state_entry.i16_next_step := ZYL_FEHLER;
						END_IF
					ELSE
						fb_ton_uz_sensor1.IN := FALSE;
					END_IF
					IF e_sensor2_ausgefahren  AND e_sensor2_eingefahren  AND st_config.b_sensor2_aktiv THEN
						fb_ton_uz_sensor2.IN := TRUE;
						IF fb_ton_uz_sensor2.Q THEN
							st_sm.b_sensor2 := TRUE;
							fb_state_entry.i16_next_step := ZYL_FEHLER;
						END_IF
					ELSE
						fb_ton_uz_sensor2.IN := FALSE;
					END_IF
				END_IF

			6:
				IF 	e_sensor1_eingefahren AND
					e_sensor2_eingefahren AND
					e_sensor3_eingefahren AND
					NOT e_sensor1_ausgefahren AND
					NOT e_sensor2_ausgefahren AND
					NOT e_sensor3_ausgefahren
					THEN
						fb_state_entry.i16_next_step := EINGEFAHREN;
				ELSE
					IF i16_betriebsart <> HAND AND st_config.b_aktiv THEN
						IF NOT e_sensor1_eingefahren OR NOT e_sensor2_eingefahren OR NOT e_sensor3_eingefahren THEN
							(* Zeitüberwachung *)
							IF fb_ton_uz_fahren.Q AND (NOT b_nockengesteuert OR b_no_gesteuert_im_norm_betrieb)THEN
								IF NOT e_sensor1_eingefahren THEN
									st_sm.b_zeit_einfahren1 := TRUE;
								END_IF
								IF NOT e_sensor2_eingefahren THEN
									st_sm.b_zeit_einfahren2 := TRUE;
								END_IF
								IF NOT e_sensor3_eingefahren THEN
									st_sm.b_zeit_einfahren3 := TRUE;
								END_IF
								fb_state_entry.i16_next_step := ZYL_FEHLER;
							(* Winkelüberwachung *)
							ELSIF uw_nocken_zylinder_einfahren AND b_nockengesteuert AND NOT b_no_gesteuert_im_norm_betrieb AND NOT b_zustand_uw_nocken_einfahren THEN
								IF NOT e_sensor1_eingefahren THEN
									st_sm.b_winkel_einfahren1 := TRUE;
								END_IF
								IF NOT e_sensor2_eingefahren THEN
									st_sm.b_winkel_einfahren2 := TRUE;
								END_IF
								IF NOT e_sensor3_eingefahren THEN
									st_sm.b_winkel_einfahren3 := TRUE;
								END_IF
								fb_state_entry.i16_next_step := ZYL_FEHLER;
							END_IF
						END_IF
					END_IF
				END_IF

				IF i16_betriebsart <> HAND AND st_config.b_aktiv THEN
					(* Überwachung auf Sensorfehler *)
					IF e_sensor1_ausgefahren  AND e_sensor1_eingefahren  AND st_config.b_sensor1_aktiv THEN
						fb_ton_uz_sensor1.IN := TRUE;
						IF fb_ton_uz_sensor1.Q THEN
							st_sm.b_sensor1 := TRUE;
							fb_state_entry.i16_next_step := ZYL_FEHLER;
						END_IF
					ELSE
						fb_ton_uz_sensor1.IN := FALSE;
					END_IF
					IF e_sensor2_ausgefahren  AND e_sensor2_eingefahren  AND st_config.b_sensor2_aktiv THEN
						fb_ton_uz_sensor2.IN := TRUE;
						IF fb_ton_uz_sensor2.Q THEN
							st_sm.b_sensor2 := TRUE;
							fb_state_entry.i16_next_step := ZYL_FEHLER;
						END_IF
					ELSE
						fb_ton_uz_sensor2.IN := FALSE;
					END_IF
					IF e_sensor3_ausgefahren  AND e_sensor3_eingefahren  AND st_config.b_sensor3_aktiv THEN
						fb_ton_uz_sensor3.IN := TRUE;
						IF fb_ton_uz_sensor3.Q THEN
							st_sm.b_sensor3 := TRUE;
							fb_state_entry.i16_next_step := ZYL_FEHLER;
						END_IF
					ELSE
						fb_ton_uz_sensor3.IN := FALSE;
					END_IF
				END_IF
		END_CASE

(*=======================================================*)
	LUFTLOS:
		IF fb_state_entry.E THEN
			a_ventil_ausfahren := FALSE;
			a_ventil_einfahren	:= FALSE;
			st_ctrl_out.b_gestoppt := FALSE;
			st_ctrl_out.b_ohne_luft := TRUE;
			st_ctrl_out.b_fehler := FALSE;
		END_IF
(*
		(* Überwachung der Sensoren *)
		CASE i16_anzahl_sensoren OF
			0:
				;

			1:
				IF b_sensor_eingefahren_vorhanden THEN
					IF st_ctrl_out.b_eingefahren AND NOT e_sensor1_eingefahren THEN
						st_sm.b_endlage1 := TRUE;
						fb_state_entry.i16_next_step := ZYL_FEHLER;
					END_IF
				ELSIF b_sensor_ausgefahren_vorhanden THEN
					IF  st_ctrl_out.b_ausgefahren AND NOT e_sensor1_ausgefahren THEN
						st_sm.b_endlage1 := TRUE;
						fb_state_entry.i16_next_step := ZYL_FEHLER;
					END_IF
				END_IF

			2:
				IF b_sensor_eingefahren_vorhanden AND b_sensor_ausgefahren_vorhanden THEN
					IF 	(st_ctrl_out.b_eingefahren AND NOT e_sensor1_eingefahren) OR
						(st_ctrl_out.b_ausgefahren AND NOT e_sensor1_ausgefahren)
						THEN
							st_sm.b_endlage1 := TRUE;
							fb_state_entry.i16_next_step := ZYL_FEHLER;
					END_IF
				ELSIF b_sensor_ausgefahren_vorhanden THEN
					IF st_ctrl_out.b_ausgefahren AND (NOT e_sensor1_ausgefahren OR NOT e_sensor2_ausgefahren) THEN
						st_sm.b_endlage1 := NOT e_sensor1_ausgefahren;
						st_sm.b_endlage2 := NOT e_sensor2_ausgefahren;
						fb_state_entry.i16_next_step := ZYL_FEHLER;
					END_IF
				ELSIF  b_sensor_eingefahren_vorhanden THEN
					IF st_ctrl_out.b_eingefahren AND (NOT e_sensor1_eingefahren OR NOT e_sensor2_eingefahren) THEN
						st_sm.b_endlage1 := NOT e_sensor1_eingefahren;
						st_sm.b_endlage2 := NOT e_sensor2_eingefahren;
						fb_state_entry.i16_next_step := ZYL_FEHLER;
					END_IF
				END_IF

			3:
				;

			4:
				IF st_ctrl_out.b_eingefahren AND (NOT e_sensor1_eingefahren OR NOT e_sensor2_eingefahren)THEN
					st_sm.b_endlage1 := NOT e_sensor1_eingefahren;
					st_sm.b_endlage2 := NOT e_sensor2_eingefahren;
					fb_state_entry.i16_next_step := ZYL_FEHLER;
				ELSIF st_ctrl_out.b_ausgefahren AND (NOT e_sensor1_ausgefahren OR NOT e_sensor2_ausgefahren)THEN
					st_sm.b_endlage1 := NOT e_sensor1_ausgefahren;
					st_sm.b_endlage2 := NOT e_sensor2_ausgefahren;
					fb_state_entry.i16_next_step := ZYL_FEHLER;
				END_IF

			6:
				IF st_ctrl_out.b_eingefahren AND (NOT e_sensor1_eingefahren OR NOT e_sensor2_eingefahren OR NOT e_sensor3_eingefahren)THEN
					st_sm.b_endlage1 := NOT e_sensor1_eingefahren;
					st_sm.b_endlage2 := NOT e_sensor2_eingefahren;
					st_sm.b_endlage3 := NOT e_sensor3_eingefahren;
					fb_state_entry.i16_next_step := ZYL_FEHLER;
				ELSIF st_ctrl_out.b_ausgefahren AND (NOT e_sensor1_ausgefahren OR NOT e_sensor2_ausgefahren OR NOT e_sensor2_ausgefahren)THEN
					st_sm.b_endlage1 := NOT e_sensor1_ausgefahren;
					st_sm.b_endlage2 := NOT e_sensor2_ausgefahren;
					st_sm.b_endlage3 := NOT e_sensor3_ausgefahren;
					fb_state_entry.i16_next_step := ZYL_FEHLER;
				END_IF
		END_CASE
*)
		(*-----------------------Weiterschaltbedingungen----------------------------*)
		CASE i16_betriebsart OF
		KEINE:
			;
		AUTO, TIPPEN, DUMMY, PSEUDO:
			IF 	(st_ctrl_in.b_ausfahren AND
				NOT st_ctrl_in.b_luftlos AND
				NOT bw_nocken_zylinder_ausfahren AND
				NOT b_ibn_zylinder_ausfahren AND
				NOT b_direkttaste_ausfahren AND
				NOT e_taste_ausfahren) OR
				(NOT st_ctrl_in.b_ausfahren AND
				NOT st_ctrl_in.b_luftlos AND
				bw_nocken_zylinder_ausfahren AND
				NOT b_ibn_zylinder_ausfahren AND
				NOT b_direkttaste_ausfahren AND
				NOT e_taste_ausfahren) OR
				(NOT st_ctrl_in.b_ausfahren AND
				NOT st_ctrl_in.b_luftlos AND
				NOT bw_nocken_zylinder_ausfahren AND
				b_ibn_zylinder_ausfahren AND
				NOT b_direkttaste_ausfahren AND
				NOT e_taste_ausfahren)
				THEN
					fb_state_entry.i16_next_step := BEWEGUNG_AUSFAHREN;

			ELSIF	(st_ctrl_in.b_einfahren AND
					NOT st_ctrl_in.b_luftlos AND
					NOT bw_nocken_zylinder_einfahren AND
					NOT b_ibn_zylinder_einfahren AND
					NOT b_direkttaste_einfahren AND
					NOT e_taste_einfahren) OR
					(NOT st_ctrl_in.b_einfahren AND
					NOT st_ctrl_in.b_luftlos AND
					bw_nocken_zylinder_einfahren AND
					NOT b_ibn_zylinder_einfahren AND
					NOT b_direkttaste_einfahren AND
					NOT e_taste_einfahren) OR
					(NOT st_ctrl_in.b_einfahren AND
					NOT st_ctrl_in.b_luftlos AND
					NOT bw_nocken_zylinder_einfahren AND
					b_ibn_zylinder_einfahren AND
					NOT b_direkttaste_einfahren AND
					NOT e_taste_einfahren)
					THEN
						fb_state_entry.i16_next_step := BEWEGUNG_EINFAHREN;
			END_IF
		HAND:
			IF	(st_visu.i16_nr_zyl_im_handbetrieb = st_config.i16_identnummer AND (st_visu.b_taste_ausfahren OR e_taste_ausfahren)) OR
				(bw_nocken_zylinder_ausfahren AND b_nockengesteuert AND b_masterachse_hand_dialog_aktiv)
				THEN
					fb_state_entry.i16_next_step := BEWEGUNG_AUSFAHREN;

			ELSIF	(st_visu.i16_nr_zyl_im_handbetrieb = st_config.i16_identnummer AND (st_visu.b_taste_einfahren OR e_taste_einfahren)) OR
					(bw_nocken_zylinder_einfahren AND b_nockengesteuert AND b_masterachse_hand_dialog_aktiv)
					THEN
						fb_state_entry.i16_next_step := BEWEGUNG_EINFAHREN;
			END_IF
		END_CASE


(*=======================================================*)
	ZYL_FEHLER:
		IF fb_state_entry.E THEN
			st_ctrl_out.b_fehler := TRUE;
			st_ctrl_out.b_eingefahren := FALSE;
			st_ctrl_out.b_ausgefahren := FALSE;
			st_ctrl_out.b_gestoppt := FALSE;
			fb_ton_quitt.IN := FALSE;
			st_visu.i16_zyl_id := st_config.i16_identnummer;
			st_visu.i16_zyl_fehlergruppe := st_config.i16_gruppe;
		END_IF

		(* Fehler wurde quittiert *)
		IF (st_ctrl_in.b_quittieren  OR b_ibn_zylinderfehler_quit ) AND NOT fb_state_entry.E THEN
			st_ctrl_out.b_fehler := FALSE;
			fb_ton_quitt.IN := TRUE;
		END_IF

		IF fb_ton_quitt.Q THEN
			fb_ton_quitt.IN := FALSE;
			fb_state_entry.i16_next_step := ZYL_INIT;
		END_IF

		(* Weiterschaltbedingungen für das Bewegen der Zylinder im Visu-Auswahlmenü im Handbetrieb, Hardwaretaster *)
		(* Zylinder einfahren im Handbetrieb über Tasten *)
		IF	i16_betriebsart = HAND AND
			st_visu.i16_nr_zyl_im_handbetrieb = st_config.i16_identnummer AND
			st_visu.b_taste_ausfahren AND
			NOT st_visu.b_taste_einfahren
			THEN
				st_ctrl_out.b_fehler := FALSE;
				st_sm.b_zeit_ausfahren1:= FALSE;
				st_sm.b_zeit_einfahren1:= FALSE;
				st_sm.b_endlage1	:= FALSE;
				st_sm.b_sensor1:= FALSE;
				st_sm.b_zeit_ausfahren2 := FALSE;
				st_sm.b_zeit_einfahren2 := FALSE;
				st_sm.b_endlage2	:= FALSE;
				st_sm.b_sensor2 := FALSE;
				st_sm.b_zeit_ausfahren3 := FALSE;
				st_sm.b_zeit_einfahren3 := FALSE;
				st_sm.b_endlage3	:= FALSE;
				st_sm.b_sensor3 := FALSE;
				st_sm.b_winkel_ausfahren1:= FALSE;
				st_sm.b_winkel_einfahren1:= FALSE;
				st_sm.b_winkel_ausfahren2 := FALSE;
				st_sm.b_winkel_einfahren2 := FALSE;
				st_sm.b_winkel_ausfahren3 := FALSE;
				st_sm.b_winkel_einfahren3 := FALSE;
				st_sm.b_zyltyp_nicht_definiert := FALSE;
				st_sm.b_reserve1:= FALSE;
				fb_state_entry.i16_next_step := BEWEGUNG_AUSFAHREN;

		(* Zylinder einfahren im Handbetrieb über Tasten *)
		ELSIF i16_betriebsart = HAND AND
			st_visu.i16_nr_zyl_im_handbetrieb = st_config.i16_identnummer AND
			st_visu.b_taste_einfahren AND
			NOT st_visu.b_taste_ausfahren
			THEN
				st_ctrl_out.b_fehler := FALSE;
				st_sm.b_zeit_ausfahren1:= FALSE;
				st_sm.b_zeit_einfahren1:= FALSE;
				st_sm.b_endlage1	:= FALSE;
				st_sm.b_sensor1:= FALSE;
				st_sm.b_zeit_ausfahren2 := FALSE;
				st_sm.b_zeit_einfahren2 := FALSE;
				st_sm.b_endlage2	:= FALSE;
				st_sm.b_sensor2 := FALSE;
				st_sm.b_zeit_ausfahren3 := FALSE;
				st_sm.b_zeit_einfahren3 := FALSE;
				st_sm.b_endlage3	:= FALSE;
				st_sm.b_sensor3 := FALSE;
				st_sm.b_winkel_ausfahren1:= FALSE;
				st_sm.b_winkel_einfahren1:= FALSE;
				st_sm.b_winkel_ausfahren2 := FALSE;
				st_sm.b_winkel_einfahren2 := FALSE;
				st_sm.b_winkel_ausfahren3 := FALSE;
				st_sm.b_winkel_einfahren3 := FALSE;
				st_sm.b_zyltyp_nicht_definiert := FALSE;
				st_sm.b_reserve1:= FALSE;
				fb_state_entry.i16_next_step := BEWEGUNG_EINFAHREN;
		END_IF

(*=======================================================*)
	DIREKT_AUSFAHREN:
		IF fb_state_entry.E THEN
			a_ventil_ausfahren := TRUE;
			a_ventil_einfahren := FALSE;
		END_IF

		IF NOT b_direkttaste_ausfahren AND NOT e_taste_ausfahren THEN
			fb_state_entry.i16_next_step := GESTOPPT;
		END_IF

(*=======================================================*)
	DIREKT_EINFAHREN:
		IF fb_state_entry.E THEN
			a_ventil_ausfahren := FALSE;
			a_ventil_einfahren := TRUE;
		END_IF

		IF NOT b_direkttaste_einfahren AND NOT e_taste_einfahren THEN
			fb_state_entry.i16_next_step := GESTOPPT;
		END_IF
END_CASE

fb_state_entry(
	i16_next_step:= ,
	i16_pos:= 2,
	s_debugtext:= ,
	E=> , 
	X=> , 
	i16_step=> ,
	i16_last_step=> );

IF st_config.b_config_fertig THEN
	(* Fehlermeldungen und Betriebsmeldungen ab dem Startindex in die globalen Meldungsarrays schreiben *)
	garr_stoermeldungen[st_config.i16_meld_startindex + 0] := st_sm.b_zeit_ausfahren1;
	garr_stoermeldungen[st_config.i16_meld_startindex + 1] := st_sm.b_zeit_einfahren1;
	garr_stoermeldungen[st_config.i16_meld_startindex + 2] := st_sm.b_endlage1;
	garr_stoermeldungen[st_config.i16_meld_startindex + 3] := st_sm.b_sensor1;
	garr_stoermeldungen[st_config.i16_meld_startindex + 4] := st_sm.b_zeit_ausfahren2;
	garr_stoermeldungen[st_config.i16_meld_startindex + 5] := st_sm.b_zeit_einfahren2;
	garr_stoermeldungen[st_config.i16_meld_startindex + 6] := st_sm.b_endlage2;
	garr_stoermeldungen[st_config.i16_meld_startindex + 7] := st_sm.b_sensor2;
	garr_stoermeldungen[st_config.i16_meld_startindex + 8] := st_sm.b_zeit_ausfahren3;
	garr_stoermeldungen[st_config.i16_meld_startindex + 9] := st_sm.b_zeit_einfahren3;
	garr_stoermeldungen[st_config.i16_meld_startindex + 10] := st_sm.b_endlage3;
	garr_stoermeldungen[st_config.i16_meld_startindex + 11] := st_sm.b_sensor3;
	garr_stoermeldungen[st_config.i16_meld_startindex + 12] := st_sm.b_winkel_ausfahren1;
	garr_stoermeldungen[st_config.i16_meld_startindex + 13] := st_sm.b_winkel_einfahren1;
	garr_stoermeldungen[st_config.i16_meld_startindex + 14] := st_sm.b_winkel_ausfahren2;
	garr_stoermeldungen[st_config.i16_meld_startindex + 15] := st_sm.b_winkel_einfahren2;
	garr_stoermeldungen[st_config.i16_meld_startindex + 16] := st_sm.b_winkel_ausfahren3;
	garr_stoermeldungen[st_config.i16_meld_startindex + 17] := st_sm.b_winkel_einfahren3;
	garr_stoermeldungen[st_config.i16_meld_startindex + 18] := st_sm.b_zyltyp_nicht_definiert;
	garr_stoermeldungen[st_config.i16_meld_startindex + 19] := st_sm.b_reserve1;
	
	garr_betriebsmeldungen[st_config.i16_meld_startindex + 0] := FALSE;
	garr_betriebsmeldungen[st_config.i16_meld_startindex + 1] := FALSE;
	garr_betriebsmeldungen[st_config.i16_meld_startindex + 2] := FALSE;
	garr_betriebsmeldungen[st_config.i16_meld_startindex + 3] := FALSE;
	garr_betriebsmeldungen[st_config.i16_meld_startindex + 4] := FALSE;
	garr_betriebsmeldungen[st_config.i16_meld_startindex + 5] := FALSE;
	garr_betriebsmeldungen[st_config.i16_meld_startindex + 6] := FALSE;
	garr_betriebsmeldungen[st_config.i16_meld_startindex + 7] := FALSE;
	garr_betriebsmeldungen[st_config.i16_meld_startindex + 8] := FALSE;
	garr_betriebsmeldungen[st_config.i16_meld_startindex + 9] := FALSE;
	garr_betriebsmeldungen[st_config.i16_meld_startindex + 10] := FALSE;
	garr_betriebsmeldungen[st_config.i16_meld_startindex + 11] := FALSE;
	garr_betriebsmeldungen[st_config.i16_meld_startindex + 12] := FALSE;
	garr_betriebsmeldungen[st_config.i16_meld_startindex + 13] := FALSE;
	garr_betriebsmeldungen[st_config.i16_meld_startindex + 14] := FALSE;
	garr_betriebsmeldungen[st_config.i16_meld_startindex + 15] := FALSE;
	garr_betriebsmeldungen[st_config.i16_meld_startindex + 16] := FALSE;
	garr_betriebsmeldungen[st_config.i16_meld_startindex + 17] := FALSE;
	garr_betriebsmeldungen[st_config.i16_meld_startindex + 18] := FALSE;
	garr_betriebsmeldungen[st_config.i16_meld_startindex + 19] := FALSE;
END_IF
END_FUNCTION_BLOCK

(* POU EPT Lib/Funktionen/WORD_TO_BOOLARRAY, ST *)
FUNCTION WORD_TO_BOOLARRAY : ARRAY[0..15] OF BOOL
VAR_INPUT
	p_inputword			: WORD;
END_VAR
VAR
	tmp_bytearray		: ARRAY[0..15] OF BOOL;
	tmp_word			: WORD;
	i16_index			: INT;
END_VAR
(* Aus einem Word, soll ein Boolarray entstehen *)
tmp_word := p_inputword;

FOR i16_index := 15 TO 0 BY -1 DO
	tmp_bytearray[i16_index] := WORD_TO_BOOL(tmp_word AND 16#8000);
	tmp_word := SHL(tmp_word, 1);
END_FOR;

WORD_TO_BOOLARRAY := tmp_bytearray; (* Rückgabewert der Funktion *)
END_FUNCTION
